// TIA Portal V20 export
DATA_BLOCK "SBK03"   // DB317
// stored: MemoryReserve 100
   VAR
      "ROLL CHANGE TOP SS.AUTO" : Bool := TRUE;
      "ROLL CHANGE BTM SS.AUTO" : Bool := TRUE;
      SPARE : Bool := FALSE;
      SPARE_1 : Bool := FALSE;
      "ROLL CHANGE TOP SS.CHANGE" : Bool := FALSE;
      "ROLL CHANGE BTM SS.CHANGE" : Bool := FALSE;
      SPARE_2 : Bool := FALSE;
      SPARE_3 : Bool := FALSE;
      "ROLL CHANGE LH IN PROGRESS" : Bool := FALSE;
      "ROLL CHANGE RH IN PROGRESS" : Bool := FALSE;
      SPARE_4 : Bool;
   END_VAR
BEGIN
END_DATA_BLOCK
